FUNCTION TryConvert_SINT_TO_TOD : BOOL
VAR_INPUT
	in : SINT;
	out : REFERENCE TO TOD;
END_VAR

IF in < DatatypeLimits.MIN_VALUE_OF_SINT_WHICH_CAN_BE_HELD_IN_A_TOD THEN
	RETURN;
END_IF

out := SINT_TO_TOD(in);
TryConvert_SINT_TO_TOD := TRUE;

END_FUNCTION

(* stored: Version 1.1.0.1, ProductVersion 3.1.4024.12
   POU TryConvert_SINT_TO_TOD: Id {bae1198c-70ad-4a1c-b1ef-eab04866db86}, SpecialFunc None *)
